TYPE ST_SerialCommSetpoints :
STRUCT
	pumpingPressureSetSetpoint : DINT;
	preHeaterTemperatureSetSetpoint : DINT ;
	separatorTemperatureSetSetpoint : DINT;
END_STRUCT
END_TYPE

(* stored: Version 1.1.0.1, ProductVersion 3.1.4024.9
   DUT ST_SerialCommSetpoints: Id {8bca8fc0-4026-4a70-8a35-64d2417d46eb} *)
